// TIA Portal V15 export
// export: Created 2018-06-03T17:22:39.4554217Z, ExportSetting WithDefaults, WithReadOnly, DisplayName Totally Integrated Automation Portal, DisplayVersion V15, DisplayName TIA Portal Openness, DisplayVersion V15, DisplayName STEP 7 Professional, DisplayVersion V15, DisplayName WinCC Professional, DisplayVersion V15
TYPE "EM_I_OUT_UDT"
// stored: CreationDate 2018-06-03T17:21:19.3788416Z, InterfaceModifiedDate 2018-06-03T17:22:01.3782438Z, IsConsistent true, IsKnowHowProtected false, LibraryConformanceStatus The object is library-conformant., ModifiedDate 2018-06-03T17:22:01.3782438Z
   STRUCT
      Request : Int;
      Command : Int;
      Pressure_SP : REAL;
      placeholder_SP_0 : Byte;   // placeholder
      placeholder_SP_1 : Byte;   // placeholder
      placeholder_SP_2 : Byte;   // placeholder
      placeholder_SP_3 : Byte;   // placeholder
      placeholder_SP_4 : Byte;   // placeholder
      placeholder_SP_5 : Byte;   // placeholder
      placeholder_SP_6 : Byte;   // placeholder
      placeholder_SP_7 : Byte;   // placeholder
      placeholder_SP_8 : Byte;   // placeholder
      placeholder_SP_9 : Byte;   // placeholder
      placeholder_SP_10 : Byte;   // placeholder
      placeholder_SP_11 : Byte;   // placeholder
      placeholder_SP_12 : Byte;   // placeholder
      placeholder_SP_13 : Byte;   // placeholder
      placeholder_SP_14 : Byte;   // placeholder
      placeholder_SP_15 : Byte;   // placeholder
      placeholder_SP_16 : Byte;   // placeholder
      placeholder_SP_17 : Byte;   // placeholder
      placeholder_SP_18 : Byte;   // placeholder
      placeholder_SP_19 : Byte;   // placeholder
      placeholder_SP_20 : Byte;   // placeholder
      placeholder_SP_21 : Byte;   // placeholder
      placeholder_SP_22 : Byte;   // placeholder
      placeholder_SP_23 : Byte;   // placeholder
      placeholder_SP_24 : Byte;   // placeholder
      placeholder_SP_25 : Byte;   // placeholder
      placeholder_SP_26 : Byte;   // placeholder
      placeholder_SP_27 : Byte;   // placeholder
      placeholder_SP_28 : Byte;   // placeholder
      placeholder_SP_29 : Byte;   // placeholder
      placeholder_SP_30 : Byte;   // placeholder
      placeholder_SP_31 : Byte;   // placeholder
      Owner : Int;
      Status : Int;
      CM_error : Bool;
      CM_error_no : DINT;
      q_bACTVIE : Bool;
      Level : REAL;
      Pressure : REAL;
      placeholder_PV_0 : Byte;   // placeholder
      placeholder_PV_1 : Byte;   // placeholder
      placeholder_PV_2 : Byte;   // placeholder
      placeholder_PV_3 : Byte;   // placeholder
      placeholder_PV_4 : Byte;   // placeholder
      placeholder_PV_5 : Byte;   // placeholder
      placeholder_PV_6 : Byte;   // placeholder
      placeholder_PV_7 : Byte;   // placeholder
      placeholder_PV_8 : Byte;   // placeholder
      placeholder_PV_9 : Byte;   // placeholder
      placeholder_PV_10 : Byte;   // placeholder
      placeholder_PV_11 : Byte;   // placeholder
      placeholder_PV_12 : Byte;   // placeholder
      placeholder_PV_13 : Byte;   // placeholder
      placeholder_PV_14 : Byte;   // placeholder
      placeholder_PV_15 : Byte;   // placeholder
      placeholder_PV_16 : Byte;   // placeholder
      placeholder_PV_17 : Byte;   // placeholder
      placeholder_PV_18 : Byte;   // placeholder
      placeholder_PV_19 : Byte;   // placeholder
   END_STRUCT;
END_TYPE
